PROGRAM MAIN
VAR
	bDin AT %I*: BOOL;	
	nAin AT %I*: INT;
	
	nSin: LREAL;
	fbton: TON;
	nTemp: REAL;
	{attribute 'TcAnalytics'}
	bDinx: BOOL;
	{attribute 'TcAnalytics'}
	nAinx: INT;
END_VAR

fbton(IN:= NOT fbton.Q,PT:= T#100MS);
IF fbton.Q THEN
	nTemp:= nTemp + 0.1;
	IF nTemp >= 3.2 THEN
		nTemp := 0;
	END_IF
END_IF
nSin := 100*SIN(nTemp);
bDinx:= bDin;
nAinx:= nAin;

END_PROGRAM

(* stored: Version 1.1.0.1, ProductVersion 3.1.4024.4
   POU MAIN: Id {2df89856-3884-4925-b50c-e9a97d85b294}, SpecialFunc None *)
